            ELSEIF n=4 THEN
                TPWrite "Go Home Position";
                rMoveHome;
                !MoveAbsJ jHomeJoint, v300, fine, tool0;
                TPWrite "Arrived Homoe Position Go to Menu";
            ELSE

                TPWrite "Go To Menu";
                WaitTime 0.3;
                GOTO gStart;

            ENDIF

        CASE 5:
            TPWrite "Go To Menu";
            WaitTime 0.3;
            GOTO gStart;
        ENDTEST

        gAuto:

    ENDPROC

    PROC rWirecut(num nRbt_No)
        bWirecut:=[FALSE,FALSE,FALSE];
        IF (sdo_Rob_1_JgHome=1 AND sdo_Rob_2_JgHome=1) OR (sdo_Rob_1_MoveHome=1 AND sdo_Rob_2_MoveHome=1) OR (sdo_Rob_1_WirecutHome=1 AND sdo_Rob_2_WirecutHome=1) THEN
        ELSE
            rMeasurementHomeCheck;
        ENDIF
        IF sdo_Rob_1_JgHome=1 AND sdo_Rob_2_JgHome=1 THEN
            bWirecut:=[TRUE,FALSE,FALSE];
            IF nRbt_No=0 OR nRbt_No=1 THEN
                Wirecut\R1;
                WaitUntil stReact{1}="WireCutOk";
                stCommand:="";
                WaitUntil stReact{1}="Ready";
            ENDIF
            IF nRbt_No=0 OR nRbt_No=2 THEN
                WireCut\R2;
                WaitUntil stReact{2}="WireCutOk";
                stCommand:="";
                WaitUntil stReact{2}="Ready";
            ENDIF
            IF nRbt_No=3 THEN
                bWireCutSync:=TRUE;
                stCommand:="WireCutR1_R2";
                WaitUntil stReact{1}="WireCutOk" AND stReact{2}="WireCutOk";
                stCommand:="";
                WaitUntil stReact{1}="Ready" AND stReact{2}="Ready";
                bWireCutSync:=FALSE;
            ENDIF
        ENDIF
        IF sdo_Rob_1_MoveHome=1 AND sdo_Rob_2_MoveHome=1 THEN
            bWirecut:=[FALSE,TRUE,FALSE];
            IF nRbt_No=0 OR nRbt_No=1 THEN
                WirecutMove\R1;
                WaitUntil stReact{1}="WireCutOk";
                stCommand:="";
                WaitUntil stReact{1}="Ready";
            ENDIF
            IF nRbt_No=0 OR nRbt_No=2 THEN
                WireCutMove\R2;
                WaitUntil stReact{2}="WireCutOk";
                stCommand:="";
                WaitUntil stReact{2}="Ready";
            ENDIF
            IF nRbt_No=3 THEN
                bWireCutSync:=TRUE;
                stCommand:="WireCutMoveR1_R2";
                WaitUntil stReact{1}="WireCutOk" AND stReact{2}="WireCutOk";
                stCommand:="";
                WaitUntil stReact{1}="Ready" AND stReact{2}="Ready";
                bWireCutSync:=FALSE;
            ENDIF
        ENDIF
        IF sdo_Rob_1_WirecutHome=1 AND sdo_Rob_2_WirecutHome=1 THEN
            bWirecut:=[FALSE,FALSE,TRUE];
            IF nRbt_No=0 OR nRbt_No=1 THEN
                WirecutShot\R1;
                WaitUntil stReact{1}="WireCutOk";
                stCommand:="";
                WaitUntil stReact{1}="Ready";
            ENDIF
            IF nRbt_No=0 OR nRbt_No=2 THEN
                WireCutShot\R2;
                WaitUntil stReact{2}="WireCutOk";
                stCommand:="";
                WaitUntil stReact{2}="Ready";
            ENDIF
            IF nRbt_No=3 THEN
                bWireCutSync:=TRUE;
                stCommand:="WireCutShotR1_R2";
                WaitUntil stReact{1}="WireCutOk" AND stReact{2}="WireCutOk";
                stCommand:="";
                WaitUntil stReact{1}="Ready" AND stReact{2}="Ready";
                bWireCutSync:=FALSE;
            ENDIF
        ENDIF
        WaitUntil stReact=["Ready","Ready","Ready"];

    ENDPROC

    PROC rWirecutShot(num nRbt_No)

        IF nRbt_No=0 OR nRbt_No=1 THEN
            WirecutShot\R1;
            WaitUntil stReact{1}="WireCutOk";
            stCommand:="";
            WaitUntil stReact{1}="Ready";
        ENDIF
        IF nRbt_No=0 OR nRbt_No=2 THEN
            WireCutShot\R2;
            WaitUntil stReact{2}="WireCutOk";
            stCommand:="";
            WaitUntil stReact{2}="Ready";
        ENDIF
        IF nRbt_No=3 THEN
            bWireCutSync:=TRUE;
            stCommand:="WireCutShotR1_R2";
            WaitUntil stReact{1}="WireCutOk" AND stReact{2}="WireCutOk";
            stCommand:="";
            WaitUntil stReact{1}="Ready" AND stReact{2}="Ready";
            bWireCutSync:=FALSE;
        ENDIF

        WaitUntil stReact=["Ready","Ready","Ready"];

    ENDPROC

    PROC rWirecutMove(num nRbt_No)

        IF nRbt_No=0 OR nRbt_No=1 THEN
            WirecutMove\R1;
            WaitUntil stReact{1}="WireCutOk";
            stCommand:="";
            WaitUntil stReact{1}="Ready";
        ENDIF
        IF nRbt_No=0 OR nRbt_No=2 THEN
            WireCutMove\R2;
            WaitUntil stReact{2}="WireCutOk";
            stCommand:="";
            WaitUntil stReact{2}="Ready";
        ENDIF
        IF nRbt_No=3 THEN
            bWireCutSync:=TRUE;
            stCommand:="WireCutMoveR1_R2";
            WaitUntil stReact{1}="WireCutOk" AND stReact{2}="WireCutOk";
            stCommand:="";
            WaitUntil stReact{1}="Ready" AND stReact{2}="Ready";
            bWireCutSync:=FALSE;
        ENDIF

        WaitUntil stReact=["Ready","Ready","Ready"];

    ENDPROC

    PROC rEdgeDataCheck()
        IF edgeStart{1}.Breadth<=0 edgeStart{1}.Breadth:=50;
        IF edgeStart{1}.Height<=0 edgeStart{1}.Height:=50;
        IF edgeStart{2}.Breadth<=0 edgeStart{2}.Breadth:=50;
        IF edgeStart{2}.Height<=0 edgeStart{2}.Height:=50;
        IF edgeEnd{1}.Breadth<=0 edgeEnd{1}.Breadth:=50;
        IF edgeEnd{1}.Height<=0 edgeEnd{1}.Height:=50;
        IF edgeEnd{2}.Breadth<=0 edgeEnd{2}.Breadth:=50;
        IF edgeEnd{2}.Height<=0 edgeEnd{2}.Height:=50;
    ENDPROC

    PROC rMoveHome_Head()

        WaitUntil stReact=["Error_Arc_Touch","Error_Arc_Touch","Error_Arc_Touch"];
        stCommand:="Error_Arc_Touch";
        WaitUntil stReact=["","",""];
        stCommand:="";
        WaitUntil stReact=["","",""];
        nErrorCmd:=1;
        ExitCycle;

    ENDPROC

    PROC rWireReplacementMode()
        VAR jointgroup jTempReadyGroup;
        VAR num nTempChangPos;
        VAR num nMaxHeight;
        !!!!!!==MoveToHome==,[
        rMeasurementHomeCheck;

        jTempReadyGroup:=MergeJgWith();
        jTempReadyGroup.JointG.extax.eax_b:=Limit(0,5300,nLimitY_Positive-nMaintenanceYPos);
        MoveJgJ MergeJgWith(\Gantry:=jTempReadyGroup.JointG),vTargetSpeed,z200;

        jTempReadyGroup.JointG.extax.eax_c:=700;
        MoveJgJ MergeJgWith(\Gantry:=jTempReadyGroup.JointG),vTargetSpeed,z200;

        RETURN ;
    ENDPROC

    PROC rArcErrorGantryDown()
        VAR jointgroup jTempReadyGroup;
        VAR num nTempGantryHeight;
        VAR num nTempPartHeightTemp;
        jTempReadyGroup:=MergeJgWith();
        nTempPartHeightTemp:=max(max(nMaxPartHeightNearArray{1},nMaxPartHeightNearArray{2}),nMaxPartHeightNearArray{3});

        nTempGantryHeight:=nHomeGantryZ-(900+nTempPartHeightTemp);
        jTempReadyGroup.JointG.extax.eax_c:=nTempGantryHeight;
        jTempReadyGroup.JointG.extax.eax_c:=Limit(0,1000,jTempReadyGroup.JointG.extax.eax_c);
        MoveJgJ MergeJgWith(\Gantry:=jTempReadyGroup.JointG),vTargetSpeed,z200;
    ENDPROC

    PROC rMeasurementHomeCheck()
        VAR jointgroup jMeasurementHomeGroup;
        VAR bool bHomeCheck:=FALSE;
        bHomeCheck:=FALSE;
        jMeasurementHomeGroup:=MergeJgWith();
        IF abs(jMeasurementHomeGroup.Joint1.robax.rax_1-jgMeasurementHome.Joint1.robax.rax_1)>1 bHomeCheck:=TRUE;
        IF abs(jMeasurementHomeGroup.Joint1.robax.rax_2-jgMeasurementHome.Joint1.robax.rax_2)>1 bHomeCheck:=TRUE;
        IF abs(jMeasurementHomeGroup.Joint1.robax.rax_3-jgMeasurementHome.Joint1.robax.rax_3)>1 bHomeCheck:=TRUE;
        IF abs(jMeasurementHomeGroup.Joint1.robax.rax_4-jgMeasurementHome.Joint1.robax.rax_4)>1 bHomeCheck:=TRUE;
        IF abs(jMeasurementHomeGroup.Joint1.robax.rax_5-jgMeasurementHome.Joint1.robax.rax_5)>1 bHomeCheck:=TRUE;
        IF abs(jMeasurementHomeGroup.Joint1.robax.rax_6-jgMeasurementHome.Joint1.robax.rax_6)>1 bHomeCheck:=TRUE;
        IF abs(jMeasurementHomeGroup.Joint2.robax.rax_1-jgMeasurementHome.Joint2.robax.rax_1)>1 bHomeCheck:=TRUE;
        IF abs(jMeasurementHomeGroup.Joint2.robax.rax_2-jgMeasurementHome.Joint2.robax.rax_2)>1 bHomeCheck:=TRUE;
        IF abs(jMeasurementHomeGroup.Joint2.robax.rax_3-jgMeasurementHome.Joint2.robax.rax_3)>1 bHomeCheck:=TRUE;
        IF abs(jMeasurementHomeGroup.Joint2.robax.rax_4-jgMeasurementHome.Joint2.robax.rax_4)>1 bHomeCheck:=TRUE;
        IF abs(jMeasurementHomeGroup.Joint2.robax.rax_5-jgMeasurementHome.Joint2.robax.rax_5)>1 bHomeCheck:=TRUE;
        IF abs(jMeasurementHomeGroup.Joint2.robax.rax_6-jgMeasurementHome.Joint2.robax.rax_6)>1 bHomeCheck:=TRUE;

        IF bHomeCheck=TRUE THEN
            rByTaskMoveToRobotHome 1;
        ELSE
            jMeasurementHomeGroup.JointG.extax.eax_c:=0;
            MoveJgJ jMeasurementHomeGroup,vTargetSpeed,fine;
        ENDIF
    ENDPROC

    PROC rjgWireCutHomeCheck()
        VAR jointgroup jWirecutHomeGroup;
        VAR bool bHomeCheck:=FALSE;
        bHomeCheck:=FALSE;
        jWirecutHomeGroup:=MergeJgWith();

        IF abs(jWirecutHomeGroup.Joint1.robax.rax_1-jgWireCutHome.Joint1.robax.rax_1)>1 bHomeCheck:=TRUE;
        IF abs(jWirecutHomeGroup.Joint1.robax.rax_2-jgWireCutHome.Joint1.robax.rax_2)>1 bHomeCheck:=TRUE;
        IF abs(jWirecutHomeGroup.Joint1.robax.rax_3-jgWireCutHome.Joint1.robax.rax_3)>1 bHomeCheck:=TRUE;
        IF abs(jWirecutHomeGroup.Joint1.robax.rax_4-jgWireCutHome.Joint1.robax.rax_4)>1 bHomeCheck:=TRUE;
        IF abs(jWirecutHomeGroup.Joint1.robax.rax_5-jgWireCutHome.Joint1.robax.rax_5)>1 bHomeCheck:=TRUE;
        IF abs(jWirecutHomeGroup.Joint1.robax.rax_6-jgWireCutHome.Joint1.robax.rax_6)>1 bHomeCheck:=TRUE;
        IF abs(jWirecutHomeGroup.Joint2.robax.rax_1-jgWireCutHome.Joint2.robax.rax_1)>1 bHomeCheck:=TRUE;
        IF abs(jWirecutHomeGroup.Joint2.robax.rax_2-jgWireCutHome.Joint2.robax.rax_2)>1 bHomeCheck:=TRUE;
        IF abs(jWirecutHomeGroup.Joint2.robax.rax_3-jgWireCutHome.Joint2.robax.rax_3)>1 bHomeCheck:=TRUE;
        IF abs(jWirecutHomeGroup.Joint2.robax.rax_4-jgWireCutHome.Joint2.robax.rax_4)>1 bHomeCheck:=TRUE;
        IF abs(jWirecutHomeGroup.Joint2.robax.rax_5-jgWireCutHome.Joint2.robax.rax_5)>1 bHomeCheck:=TRUE;
        IF abs(jWirecutHomeGroup.Joint2.robax.rax_6-jgWireCutHome.Joint2.robax.rax_6)>1 bHomeCheck:=TRUE;

        IF bHomeCheck=TRUE THEN
            rByTaskMoveToRobotHome 2;
        ELSE
            jWirecutHomeGroup.JointG.extax.eax_c:=0;
            MoveJgJ jWirecutHomeGroup,vTargetSpeed,fine;
        ENDIF
    ENDPROC

    PROC rByTaskMoveToRobotHome(num nHomeNo)
        VAR jointgroup jgEmptyTarget;
        VAR jointtarget jTempG;
        VAR num ntemp;

        stCommand:="checkpos";
        waituntil stReact=["checkposok","checkposok","checkposok"];
        stCommand:="";
        waituntil stReact=["Ready","Ready","Ready"];

        jgEmptyTarget.Joint1:=CJointT(\TaskName:="T_Rob1");
        jgEmptyTarget.Joint2:=CJointT(\TaskName:="T_Rob2");
        jgEmptyTarget.JointG:=CJointT(\TaskName:="T_Rob1");
        jgEmptyTarget.JointG.extax.eax_c:=0;
        MoveJgJ jgEmptyTarget,vTargetSpeed,fine;

        jgEmptyTarget.Joint1.robax.rax_2:=-90;
        jgEmptyTarget.Joint1.robax.rax_3:=55;
        jgEmptyTarget.Joint2.robax.rax_2:=-90;
        jgEmptyTarget.Joint2.robax.rax_3:=55;
        MoveJgJ jgEmptyTarget,vTargetSpeed,fine;

        jgEmptyTarget.Joint1.robax.rax_5:=0;
        jgEmptyTarget.Joint2.robax.rax_5:=0;
        MoveJgJ jgEmptyTarget,vTargetSpeed,fine;
        IF nHomeNo=1 THEN
            jgEmptyTarget.Joint1.robax.rax_1:=jgMeasurementHome.Joint1.robax.rax_1;
            jgEmptyTarget.Joint2.robax.rax_1:=jgMeasurementHome.Joint2.robax.rax_1;
        ELSEIF nHomeNo=2 THEN
            jgEmptyTarget.Joint1.robax.rax_1:=jgWireCutHome.Joint1.robax.rax_1;
            jgEmptyTarget.Joint2.robax.rax_1:=jgWireCutHome.Joint2.robax.rax_1;
        ENDIF
        jgEmptyTarget.JointG.extax.eax_d:=0;
        MoveJgJ jgEmptyTarget,vTargetSpeed,fine;

        jgEmptyTarget.Joint1:=CJointT(\TaskName:="T_Rob1");
        jgEmptyTarget.Joint2:=CJointT(\TaskName:="T_Rob2");
        jgEmptyTarget.JointG:=CJointT(\TaskName:="T_Rob1");
        IF nHomeNo=1 THEN
            jgEmptyTarget.Joint1.robax:=jgMeasurementHome.Joint1.robax;
            jgEmptyTarget.Joint2.robax:=jgMeasurementHome.Joint2.robax;
        ELSEIF nHomeNo=2 THEN
            jgEmptyTarget.Joint1.robax:=jgWireCutHome.Joint1.robax;
            jgEmptyTarget.Joint2.robax:=jgWireCutHome.Joint2.robax;
        ENDIF
        MoveJgJ jgEmptyTarget,vTargetSpeed,fine;

        RETURN ;
    ENDPROC

     PROC rWarm_Up()
        VAR jointgroup jgWarm_Up;
        VAR speeddata vWarmUp_Speed:=[0,0,0,0];
        VAR num i:=0;
        VAR num nWarmUp_Distance_X;
        VAR num nWarmUp_Distance_Y;
        VAR num nWarmUp_Distance_Z;
        VAR num nWarmUp_Distance_R;

        FOR i FROM 1 TO nWarmUp_Count*2 DO
            nWarmUp_Distance_X:=nWarmUp_Distance;
            nWarmUp_Distance_Y:=nWarmUp_Distance;
            nWarmUp_Distance_Z:=nWarmUp_Distance;
            nWarmUp_Distance_R:=(nWarmUp_Distance/488)*57.2958;
            vWarmUp_Speed:=[nWarmUp_Speed,nWarmUp_Speed*(nWarmUp_Speed/488)*(180/pi),nWarmUp_Speed,nWarmUp_Speed*(nWarmUp_Speed/488)*(180/pi)];
            jgWarm_Up:=MergeJgWith();
            IF jgWarm_Up.JointG.extax.eax_a+nWarmUp_Distance_X<nLimitX_Negative OR jgWarm_Up.JointG.extax.eax_a+nWarmUp_Distance_X>nLimitX_Positive THEN
                jgWarm_Up.JointG.extax.eax_a:=jgWarm_Up.JointG.extax.eax_a-nWarmUp_Distance_X;
                jgWarm_Up.JointG.extax.eax_f:=jgWarm_Up.JointG.extax.eax_f-nWarmUp_Distance_X;
            ELSE
                jgWarm_Up.JointG.extax.eax_a:=jgWarm_Up.JointG.extax.eax_a+nWarmUp_Distance_X;
                jgWarm_Up.JointG.extax.eax_f:=jgWarm_Up.JointG.extax.eax_f+nWarmUp_Distance_X;
            ENDIF

            IF jgWarm_Up.JointG.extax.eax_b+nWarmUp_Distance_Y<nLimitY_Negative OR jgWarm_Up.JointG.extax.eax_b+nWarmUp_Distance_Y>nLimitY_Positive THEN
                jgWarm_Up.JointG.extax.eax_b:=jgWarm_Up.JointG.extax.eax_b-nWarmUp_Distance_Y;
            ELSE
                jgWarm_Up.JointG.extax.eax_b:=jgWarm_Up.JointG.extax.eax_b+nWarmUp_Distance_Y;
            ENDIF

            IF jgWarm_Up.JointG.extax.eax_c+nWarmUp_Distance_Z<nLimitZ_Negative OR jgWarm_Up.JointG.extax.eax_c+nWarmUp_Distance_Z>750 THEN
                jgWarm_Up.JointG.extax.eax_c:=jgWarm_Up.JointG.extax.eax_c-nWarmUp_Distance_Z;
            ELSE
                jgWarm_Up.JointG.extax.eax_c:=jgWarm_Up.JointG.extax.eax_c+nWarmUp_Distance_Z;
            ENDIF

            IF jgWarm_Up.JointG.extax.eax_d+nWarmUp_Distance_R<nLimitR_Negative OR jgWarm_Up.JointG.extax.eax_d+nWarmUp_Distance_R>nLimitR_Positive THEN
                jgWarm_Up.JointG.extax.eax_d:=jgWarm_Up.JointG.extax.eax_d-nWarmUp_Distance_R;
            ELSE
                jgWarm_Up.JointG.extax.eax_d:=jgWarm_Up.JointG.extax.eax_d+nWarmUp_Distance_R;
            ENDIF

            jgWarm_Up.JointG.extax.eax_a:=Limit(nLimitX_Negative,nLimitX_Positive,jgWarm_Up.JointG.extax.eax_a);
            jgWarm_Up.JointG.extax.eax_b:=Limit(nLimitY_Negative,nLimitY_Positive,jgWarm_Up.JointG.extax.eax_b);
            jgWarm_Up.JointG.extax.eax_c:=Limit(nLimitZ_Negative,750,jgWarm_Up.JointG.extax.eax_c);
            jgWarm_Up.JointG.extax.eax_d:=Limit(nLimitR_Negative,nLimitR_Positive,jgWarm_Up.JointG.extax.eax_d);
            jgWarm_Up.JointG.extax.eax_f:=Limit(nLimitX_Negative,nLimitX_Positive,jgWarm_Up.JointG.extax.eax_f);

            MoveJgJ MergeJgWith(\Gantry:=jgWarm_Up.JointG),vWarmUp_Speed,fine;
            nWarmUp_Distance:=nWarmUp_Distance*(-1);
        ENDFOR
        RETURN ;
    ENDPROC
ENDMODULE
